(*
SPDX-FileCopyrightText: © 2026 Oleksandr Tiutyk <trofimich@gmail.com>
SPDX-License-Identifier: MIT
License: https://opensource.org/license/mit
*)

(*!
<summary>Provides the object's application or diagnostic name.</summary>
<description>
The name is not guaranteed to be a unique object identifier.
</description>
*)

INTERFACE INamed EXTENDS IObject

(*!
<summary>Returns a borrowed, read-only view of the name without copying its storage.</summary>
<description>
Read-only is a usage contract: callers must not write through the returned reference. The reference requires a
live provider and is not a snapshot; copy the value when an independent name is needed.
</description>
*)

{attribute 'monitoring' := 'call'}
PROPERTY Name : REFERENCE TO WSTRING
GET
END_GET
END_PROPERTY

END_INTERFACE

(* stored: Version 1.1.0.1
   Itf INamed: Id {494b9ae3-adc0-4a55-b03f-05645ae69372}
   Property Name: Id {72c457aa-a371-4a9a-b527-076a57a0f56a}
   Get Get: Id {7c0fd7b8-0488-427f-960f-92755ac998ce} *)
